INTERFACE IGenericPredicate EXTENDS IObject

METHOD Compare : BOOL
VAR_IN_OUT CONSTANT
	objectToCompare : GENERIC_VALUE; 
END_VAR
END_METHOD

END_INTERFACE

(* stored: Version 1.1.0.1
   Itf IGenericPredicate: Id {2d6a38ba-260b-4d26-a5bc-9bd5e6db19e8}
   Method Compare: Id {481953a6-7290-46b0-ac08-ad672ed4bf66} *)
